(* Schneider Machine Expert - Basic project Water Level Controller (WLC), file version 1.7.0.0 *)
(* ProjectInformations: Name=New project *)

HARDWARE
  Cpu 0: TM221ME32TK
  EthernetConfiguration: NetworkName=M221, IpAllocationMode=FixedAddress, IpAddress=0.0.0.0, SubnetMask=0.0.0.0
  SerialLineConfiguration: Baud=Baud19200, Parity=ParityEven, DataBits=DataBits8, StopBits=StopBits1, PhysicalMedium=PhysicalMediumRs485, TransmissionMode=TransmissionModeModbusRtu, SlaveId=1, Addressing=SlaveAddressing
  MastTask: UsePeriodScanMode=false, PeriodScan=100
  FastTask: Period=255
  CpuBehavior: StartingMode=StartAsPreviousState, AutoSaveRamOnEeprom=true, WatchdogPeriod=250

SYMBOLS  (address, symbol, comment, settings)
  %I0.0       "Manual"
  %I0.1       "Auto"
  %I0.2       "LSLL"
  %I0.3       "LSL"
  %I0.4       "LSH"
  %I0.5       "LSHH"
  %I0.6       "S1"
  %I0.7       "S2"
  %I0.8       "S3"
  %Q0.0       "P1"
  %Q0.1       "P2"
  %Q0.2       "SOV"

POU New POU
  (* SectionNumber=1 *)

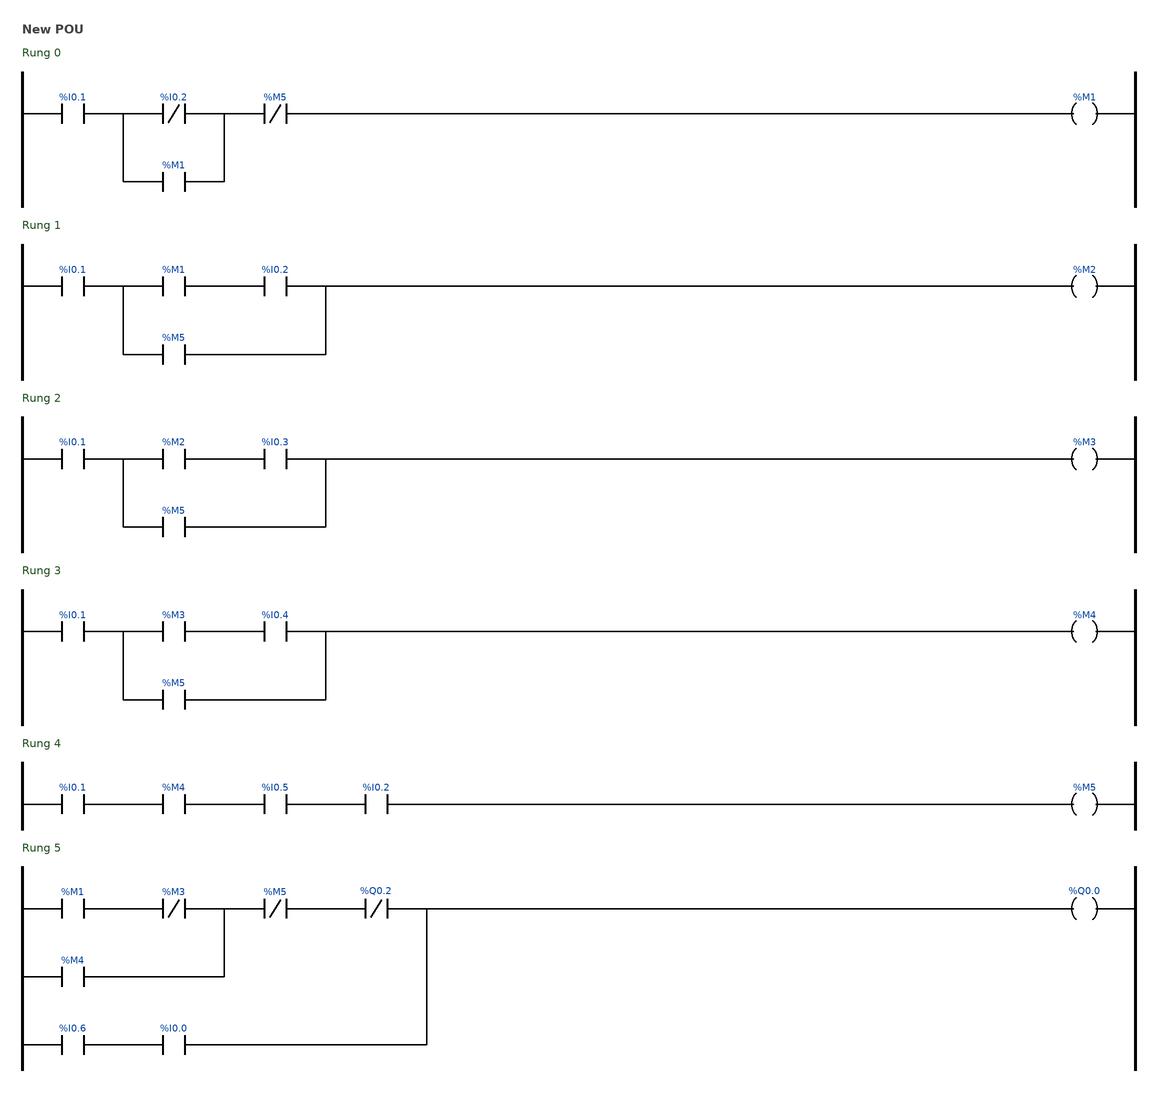

// Rung 0
  LD %I0.1
  AND(N %I0.2
  OR %M1
  )
  ANDN %M5
  ST %M1
  // as ST:
  //   %M1 := %I0.1 AND (NOT %I0.2 OR %M1) AND NOT %M5;

// Rung 1
  LD %I0.1
  AND( %M1
  AND %I0.2
  OR %M5
  )
  ST %M2
  // as ST:
  //   %M2 := %I0.1 AND (%M1 AND %I0.2 OR %M5);

// Rung 2
  LD %I0.1
  AND( %M2
  AND %I0.3
  OR %M5
  )
  ST %M3
  // as ST:
  //   %M3 := %I0.1 AND (%M2 AND %I0.3 OR %M5);

// Rung 3
  LD %I0.1
  AND( %M3
  AND %I0.4
  OR %M5
  )
  ST %M4
  // as ST:
  //   %M4 := %I0.1 AND (%M3 AND %I0.4 OR %M5);

// Rung 4
  LD %I0.1
  AND %M4
  AND %I0.5
  AND %I0.2
  ST %M5
  // as ST:
  //   %M5 := %I0.1 AND %M4 AND %I0.5 AND %I0.2;

// Rung 5
  LD %M1
  ANDN %M3
  OR %M4
  ANDN %M5
  ANDN %Q0.2
  OR( %I0.6
  AND %I0.0
  )
  ST %Q0.0
  // as ST:
  //   %Q0.0 := (%M1 AND NOT %M3 OR %M4) AND NOT %M5 AND NOT %Q0.2 OR %I0.6 AND %I0.0;

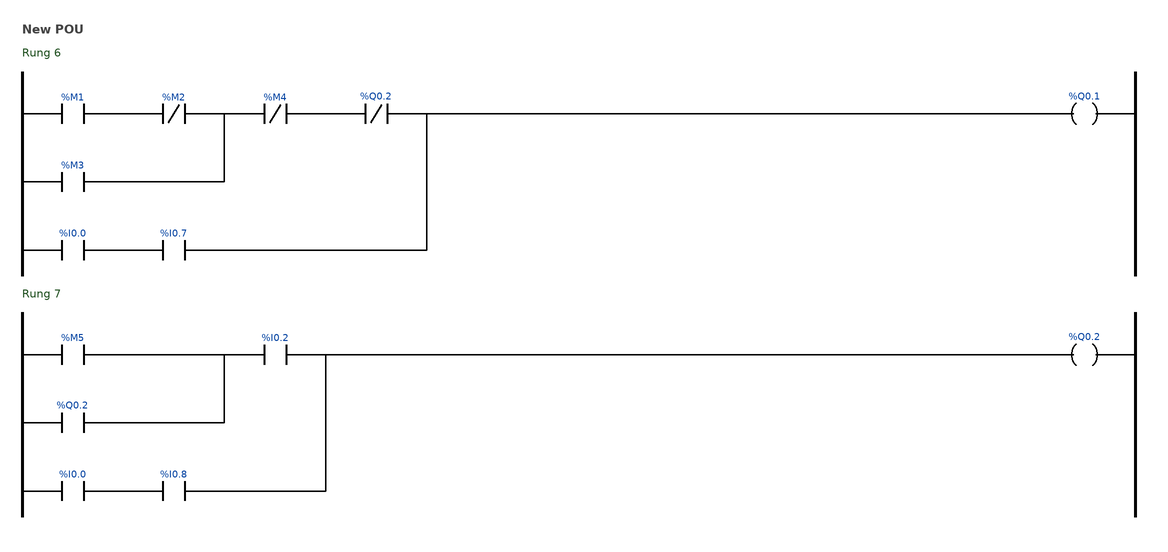

// Rung 6
  LD %M1
  ANDN %M2
  OR %M3
  ANDN %M4
  ANDN %Q0.2
  OR( %I0.0
  AND %I0.7
  )
  ST %Q0.1
  // as ST:
  //   %Q0.1 := (%M1 AND NOT %M2 OR %M3) AND NOT %M4 AND NOT %Q0.2 OR %I0.0 AND %I0.7;

// Rung 7
  LD %M5
  OR %Q0.2
  AND %I0.2
  OR( %I0.0
  AND %I0.8
  )
  ST %Q0.2
  // as ST:
  //   %Q0.2 := (%M5 OR %Q0.2) AND %I0.2 OR %I0.0 AND %I0.8;
